(*
SPDX-FileCopyrightText: © 2026 Oleksandr Tiutyk <trofimich@gmail.com>
SPDX-License-Identifier: MIT
License: https://opensource.org/license/mit
*)

{attribute 'qualified_only'}
VAR_GLOBAL
	Name : STRING := 'TOF_Samples';
END_VAR

(* stored: Version 1.1.0.1
   GVL CurrentNamespace: Id {ca939c29-8d6f-49b1-a037-35523be7f11f} *)
